// TIA Portal V16 export
// export: Created 2023-10-30T22:43:55.7598757Z, ExportSetting WithDefaults, DisplayName Totally Integrated Automation Portal, DisplayVersion V16, DisplayName TIA Portal Version Control Interface, DisplayVersion V16, DisplayName TIA Portal Openness, DisplayVersion V16, DisplayName SINAMICS Startdrive Advanced, DisplayVersion V16, DisplayName SINAMICS Startdrive G130, G150, S120, S150, SINAMICS MV, S210, DisplayVersion V16, DisplayName SINAMICS Startdrive G110M, G120, G120C, G120D, G120P, DisplayVersion V16, DisplayName STEP 7 Professional, DisplayVersion V16, DisplayName STEP 7 Safety, DisplayVersion V16, DisplayName WinCC Professional, DisplayVersion V16
DATA_BLOCK "Filtro_Promedio_DB"   // DB21
VERSION : 0.1
// stored: AutoNumber true, DBAccessibleFromOPCUA true, InstanceOfName Filtro_Promedio, InstanceOfType FB
"Filtro_Promedio"
   // VAR_INPUT
   //    N : Int;
   //    "D.IN" : Real;
   // END_VAR
   // VAR_OUTPUT
   //    "D.OUT" : Real;
   // END_VAR
   // VAR
   //    D : Array[0..100] of Real;
   //    I : Int;
   //    J : Int;
   //    "D.Sum" : Real;
   // END_VAR
BEGIN
END_DATA_BLOCK
